GLOBALCONSTANTS DefaultPool_TECU_Numeric (* Numeric object pool constants (ID, Scale, Offset, Decimals) *)
  PACKAGE Uebungen::const::UT::TECU;
  VAR_GLOBAL CONSTANT
    OutputNumber_Wheel_based_machine_speed_km_h_N : logiBUS::utils::conversion::phys::NumericObjectPool_S := (u16ObjId := 12000, r32Scale := 0.0036, i32Offset := 0, u8Decimals := 1);
    OutputNumber_Wheel_based_machine_speed_m_s_N : logiBUS::utils::conversion::phys::NumericObjectPool_S := (u16ObjId := 12001, r32Scale := 0.001, i32Offset := 0, u8Decimals := 1);
    OutputNumber_Ground_based_machine_speed_km_h_N : logiBUS::utils::conversion::phys::NumericObjectPool_S := (u16ObjId := 12002, r32Scale := 0.0036, i32Offset := 0, u8Decimals := 1);
    OutputNumber_Ground_based_machine_speed_m_s_N : logiBUS::utils::conversion::phys::NumericObjectPool_S := (u16ObjId := 12003, r32Scale := 0.001, i32Offset := 0, u8Decimals := 1);
    OutputNumber_Wheel_based_machine_distance_km_N : logiBUS::utils::conversion::phys::NumericObjectPool_S := (u16ObjId := 12004, r32Scale := 0.000001, i32Offset := 0, u8Decimals := 1);
    OutputNumber_Wheel_based_machine_distance_m_N : logiBUS::utils::conversion::phys::NumericObjectPool_S := (u16ObjId := 12005, r32Scale := 0.001, i32Offset := 0, u8Decimals := 1);
    OutputNumber_Rear_PTO_output_shaft_speed_N : logiBUS::utils::conversion::phys::NumericObjectPool_S := (u16ObjId := 12006, r32Scale := 0.125, i32Offset := 0, u8Decimals := 1);
    OutputNumber_TECU_Speed_WBSD_N : logiBUS::utils::conversion::phys::NumericObjectPool_S := (u16ObjId := 12024, r32Scale := 0.001, i32Offset := 0, u8Decimals := 1);
    OutputNumber_TECU_Speed_GBSD_N : logiBUS::utils::conversion::phys::NumericObjectPool_S := (u16ObjId := 12025, r32Scale := 0.001, i32Offset := 0, u8Decimals := 1);
    OutputNumber_TECU_Speed_MSS_N : logiBUS::utils::conversion::phys::NumericObjectPool_S := (u16ObjId := 12026, r32Scale := 0.001, i32Offset := 0, u8Decimals := 1);
    OutputNumber_TECU_Speed_VDS_N : logiBUS::utils::conversion::phys::NumericObjectPool_S := (u16ObjId := 12027, r32Scale := 0.001, i32Offset := 0, u8Decimals := 1);
    OutputNumber_TECU_Speed_COGSOG_N : logiBUS::utils::conversion::phys::NumericObjectPool_S := (u16ObjId := 12028, r32Scale := 0.001, i32Offset := 0, u8Decimals := 1);
    OutputNumber_TECU_FHS_Position_N : logiBUS::utils::conversion::phys::NumericObjectPool_S := (u16ObjId := 12029, r32Scale := 0.4, i32Offset := 0, u8Decimals := 1);
    OutputNumber_TECU_RHS_Position_N : logiBUS::utils::conversion::phys::NumericObjectPool_S := (u16ObjId := 12030, r32Scale := 0.4, i32Offset := 0, u8Decimals := 1);
    OutputNumber_TECU_FHS_Force_N : logiBUS::utils::conversion::phys::NumericObjectPool_S := (u16ObjId := 12031, r32Scale := 1.0, i32Offset := 0, u8Decimals := 0);
    OutputNumber_TECU_RHS_Force_N : logiBUS::utils::conversion::phys::NumericObjectPool_S := (u16ObjId := 12032, r32Scale := 1.0, i32Offset := 0, u8Decimals := 0);
    OutputNumber_TECU_FHS_Draft_N : logiBUS::utils::conversion::phys::NumericObjectPool_S := (u16ObjId := 12033, r32Scale := 1.0, i32Offset := 0, u8Decimals := 0);
    OutputNumber_TECU_RHS_Draft_N : logiBUS::utils::conversion::phys::NumericObjectPool_S := (u16ObjId := 12034, r32Scale := 1.0, i32Offset := 0, u8Decimals := 0);
    OutputNumber_TECU_FPTO_Speed_N : logiBUS::utils::conversion::phys::NumericObjectPool_S := (u16ObjId := 12035, r32Scale := 0.125, i32Offset := 0, u8Decimals := 1);
    OutputNumber_TECU_RPTO_Speed_N : logiBUS::utils::conversion::phys::NumericObjectPool_S := (u16ObjId := 12036, r32Scale := 0.125, i32Offset := 0, u8Decimals := 1);
    OutputNumber_TECU_FPTO_SpeedSet_N : logiBUS::utils::conversion::phys::NumericObjectPool_S := (u16ObjId := 12037, r32Scale := 0.125, i32Offset := 0, u8Decimals := 1);
    OutputNumber_TECU_RPTO_SpeedSet_N : logiBUS::utils::conversion::phys::NumericObjectPool_S := (u16ObjId := 12038, r32Scale := 0.125, i32Offset := 0, u8Decimals := 1);
    NumberVariable_Wheel_based_machine_speed_N : logiBUS::utils::conversion::phys::NumericObjectPool_S := (u16ObjId := 21000, r32Scale := 0.001, i32Offset := 0, u8Decimals := 1);
    NumberVariable_Ground_based_machine_speed_N : logiBUS::utils::conversion::phys::NumericObjectPool_S := (u16ObjId := 21001, r32Scale := 0.001, i32Offset := 0, u8Decimals := 1);
    NumberVariable_Wheel_based_machine_distance_N : logiBUS::utils::conversion::phys::NumericObjectPool_S := (u16ObjId := 21002, r32Scale := 0.000001, i32Offset := 0, u8Decimals := 1);
    NumberVariable_Rear_PTO_output_shaft_speed_N : logiBUS::utils::conversion::phys::NumericObjectPool_S := (u16ObjId := 21003, r32Scale := 0.125, i32Offset := 0, u8Decimals := 1);
    NumberVariable_TECU_Speed_WBSD_N : logiBUS::utils::conversion::phys::NumericObjectPool_S := (u16ObjId := 21024, r32Scale := 0.001, i32Offset := 0, u8Decimals := 1);
    NumberVariable_TECU_Speed_GBSD_N : logiBUS::utils::conversion::phys::NumericObjectPool_S := (u16ObjId := 21025, r32Scale := 0.001, i32Offset := 0, u8Decimals := 1);
    NumberVariable_TECU_Speed_MSS_N : logiBUS::utils::conversion::phys::NumericObjectPool_S := (u16ObjId := 21026, r32Scale := 0.001, i32Offset := 0, u8Decimals := 1);
    NumberVariable_TECU_Speed_VDS_N : logiBUS::utils::conversion::phys::NumericObjectPool_S := (u16ObjId := 21027, r32Scale := 0.001, i32Offset := 0, u8Decimals := 1);
    NumberVariable_TECU_Speed_COGSOG_N : logiBUS::utils::conversion::phys::NumericObjectPool_S := (u16ObjId := 21028, r32Scale := 0.001, i32Offset := 0, u8Decimals := 1);
    NumberVariable_TECU_FHS_Position_N : logiBUS::utils::conversion::phys::NumericObjectPool_S := (u16ObjId := 21029, r32Scale := 0.4, i32Offset := 0, u8Decimals := 1);
    NumberVariable_TECU_RHS_Position_N : logiBUS::utils::conversion::phys::NumericObjectPool_S := (u16ObjId := 21030, r32Scale := 0.4, i32Offset := 0, u8Decimals := 1);
    NumberVariable_TECU_FHS_Force_N : logiBUS::utils::conversion::phys::NumericObjectPool_S := (u16ObjId := 21031, r32Scale := 1.0, i32Offset := 0, u8Decimals := 0);
    NumberVariable_TECU_RHS_Force_N : logiBUS::utils::conversion::phys::NumericObjectPool_S := (u16ObjId := 21032, r32Scale := 1.0, i32Offset := 0, u8Decimals := 0);
    NumberVariable_TECU_FHS_Draft_N : logiBUS::utils::conversion::phys::NumericObjectPool_S := (u16ObjId := 21033, r32Scale := 1.0, i32Offset := 0, u8Decimals := 0);
    NumberVariable_TECU_RHS_Draft_N : logiBUS::utils::conversion::phys::NumericObjectPool_S := (u16ObjId := 21034, r32Scale := 1.0, i32Offset := 0, u8Decimals := 0);
    NumberVariable_TECU_FPTO_Speed_N : logiBUS::utils::conversion::phys::NumericObjectPool_S := (u16ObjId := 21035, r32Scale := 0.125, i32Offset := 0, u8Decimals := 1);
    NumberVariable_TECU_RPTO_Speed_N : logiBUS::utils::conversion::phys::NumericObjectPool_S := (u16ObjId := 21036, r32Scale := 0.125, i32Offset := 0, u8Decimals := 1);
    NumberVariable_TECU_FPTO_SpeedSet_N : logiBUS::utils::conversion::phys::NumericObjectPool_S := (u16ObjId := 21037, r32Scale := 0.125, i32Offset := 0, u8Decimals := 1);
    NumberVariable_TECU_RPTO_SpeedSet_N : logiBUS::utils::conversion::phys::NumericObjectPool_S := (u16ObjId := 21038, r32Scale := 0.125, i32Offset := 0, u8Decimals := 1);
  END_VAR
END_GLOBALCONSTANTS
(* other elements stored in the file *)
(* ACHTUNG: 'NumberVariable_Wheel_based_machine_speed' wird von mehreren Widgets mit unterschiedlicher Skalierung gebunden - 'OutputNumber_Wheel_based_machine_speed_km_h' (scale=0.0036 offset=0 decimals=1) vs. 'OutputNumber_Wheel_based_machine_speed_m_s' (scale=0.001 offset=0 decimals=1). Es gilt die Skalierung mit dem kleinsten |Scale|, alle Widgets muessen dieselbe Skalierung haben. *)
(* ACHTUNG: 'NumberVariable_Ground_based_machine_speed' wird von mehreren Widgets mit unterschiedlicher Skalierung gebunden - 'OutputNumber_Ground_based_machine_speed_km_h' (scale=0.0036 offset=0 decimals=1) vs. 'OutputNumber_Ground_based_machine_speed_m_s' (scale=0.001 offset=0 decimals=1). Es gilt die Skalierung mit dem kleinsten |Scale|, alle Widgets muessen dieselbe Skalierung haben. *)
(* ACHTUNG: 'NumberVariable_Wheel_based_machine_distance' wird von mehreren Widgets mit unterschiedlicher Skalierung gebunden - 'OutputNumber_Wheel_based_machine_distance_km' (scale=1e-06 offset=0 decimals=1) vs. 'OutputNumber_Wheel_based_machine_distance_m' (scale=0.001 offset=0 decimals=1). Es gilt die Skalierung mit dem kleinsten |Scale|, alle Widgets muessen dieselbe Skalierung haben. *)
